INTERFACE I_AlarmContext

PROPERTY Acknowledge : BOOL
GET
END_GET
END_PROPERTY

METHOD AddNewAlarm : DINT
VAR_INPUT
	iAlarm : I_Alarm;
END_VAR
END_METHOD

METHOD EnableAcknowledge : BOOL
VAR_INPUT
	nAlarmContextId		: DINT;
	bCanByAcknowledged	: BOOL;
END_VAR
END_METHOD

PROPERTY IsAlarmBufferFull : BOOL
GET
END_GET
END_PROPERTY

METHOD RemoveAlarm : BOOL
VAR_INPUT
	nAlarmContextId : DINT;
END_VAR
END_METHOD

PROPERTY SelectedAlarmContextId : DINT
GET
END_GET
END_PROPERTY

END_INTERFACE

(* stored: Version 1.1.0.1, ProductVersion 3.1.4024.15
   Itf I_AlarmContext: Id {771b6988-0709-4c75-8e82-dfd8ec524245}
   Property Acknowledge: Id {07d16865-68b4-46b2-a8d9-76825b9370a5}
   Get Get: Id {d228de9d-2310-47c2-8e08-d20f5531e0db}
   Method AddNewAlarm: Id {10388e2c-3ad8-4a45-a43e-5b3ecc097722}
   Method EnableAcknowledge: Id {e79202b3-4d68-4058-a378-96b1778c659e}
   Property IsAlarmBufferFull: Id {c4af422c-0c7b-4be1-8948-4f10649d7b82}
   Get Get: Id {e278ec41-7153-41c9-9a6a-328637f73f52}
   Method RemoveAlarm: Id {70ea4550-008d-4922-b512-a097b6f46f95}
   Property SelectedAlarmContextId: Id {fb8f4d44-0eee-4911-8615-e4224116402a}
   Get Get: Id {b09fa67e-a690-42ac-b103-1d2b25eab725} *)
